// TwinCAT 3 PLC project InovanceDemo
// ProgramVersion: 3.1.4024.0
// libraries:
//   Tc2_MC2, * (Beckhoff Automation GmbH)
//   Tc2_Standard, * (Beckhoff Automation GmbH)
//   Tc2_System, * (Beckhoff Automation GmbH)
//   Tc3_Module, * (Beckhoff Automation GmbH)
// project tree:
//   DUTs/ MoveState.TcDUT
//   / PlcTask.TcTTO
//   POUs/ MAIN.TcPOU
// real-time tasks:
//   TASK PlcTask: cycle T#10ms, priority 20, ADS port 350
// motion (NC):
//   TASK NC-Task 1 SAF: cycle T#2ms, priority 4, ADS port 501
//   TASK NC-Task 1 SVB: cycle T#10ms, priority 8, ADS port 511
//   AXIS Axis 1 (id 1)
//     Velo: SlowManual=500
//     PositionAreaControl: Enable=false
//     TargetPosControl: Enable=false
//     OtherSettings: AllowMotionCmdToSlave=true
//     encoder EncType=1
//       EncPara: ScaleFactorNumerator=1.788e-05
//     drive DrvType=5
//       Analog: TorqueSetpointScale=10, ScaleFactorActTorque=0.1
//       TimeComp: TaskDelayCycles=1
//     controller CtrType=1
//       CtrPara: PriorControlFactor=1
//         PosDiffControl: Enable=false
//         Observer: BandWidth=20
// I/O:
//   DEVICE Device 3 (EtherCAT), AmsNetId 192.168.148.33.4.1
//     Drive 1 (InoSV660N) [SV660_1Axis_00915] (disabled)
// variable links:
//   InovanceDemo/InovanceDemo Instance <-> NC-Task 1 SAF/Axes/Axis 1
//     PlcTask Inputs/MAIN.Axis1.NcToPlc <-> Outputs/ToPlc
//     PlcTask Outputs/MAIN.Axis1.PlcToNc <-> Inputs/FromPlc

CONFIGURATION InovanceDemo
    RESOURCE PLC ON TwinCAT3
        TASK PlcTask(INTERVAL := T#10ms, PRIORITY := 20);
        PROGRAM MAIN WITH PlcTask : MAIN;
    END_RESOURCE
END_CONFIGURATION

// ---- DUTs/MoveState.TcDUT
TYPE MoveState :
(
	MOVE_INIT ,
	MOVE_ENABLE ,
	MOVE_MOVEFORWARD ,
	MOVE_MOVEBACKWARD ,
	MOVE_ERROR ,
	MOVE_RESET
)UDINT;
END_TYPE

// ---- POUs/MAIN.TcPOU
PROGRAM MAIN
VAR
	Axis1 : AXIS_REF;
	
	PowerAxis1 : MC_Power;
	PowerAxis1Out : ST_McOutputs;
	
	ResetAxis1 : MC_Reset;
	ResetAxis1Out : ST_McOutputs;
	
	MoveAxis1 : MC_MoveAbsolute();
	MoveAxis2 : MC_MoveAbsolute;
	MoveAbsolute1 : ST_McOutputs;
	MoveAbsolute2 : ST_McOutputs;
	
	
	state : MoveState;
	
END_VAR


	(* update the axis status at the beginning of each cycle *)
	Axis1();
	
	(* move axis using a state machine *)
	CASE state OF
		
		MOVE_INIT :
			MoveAxis1.Execute := FALSE;
			MoveAxis2.Execute := FALSE;
			ResetAxis1.Execute := FALSE;
			state := MOVE_ENABLE;
		
		MOVE_ENABLE:
			PowerAxis1.Enable := TRUE;
			PowerAxis1.Enable_Positive := TRUE;
			PowerAxis1.Enable_Negative := TRUE;
			IF PowerAxis1.Status THEN
				state := MOVE_MOVEFORWARD;
			ELSIF PowerAxis1.Error THEN	
				state := MOVE_ERROR;
			END_IF
		MOVE_MOVEFORWARD:
			MoveAxis1.Execute := TRUE;
			MoveAxis1.Position := 500;
			MoveAxis1.Velocity := 500;
			
			IF MoveAxis1.Error THEN
				state := MOVE_ERROR;
			ELSIF MoveAxis1.Done THEN
				MoveAxis1.Execute := FALSE;
				state := MOVE_MOVEBACKWARD;
			END_IF
			
		MOVE_MOVEBACKWARD:
			MoveAxis1.Execute := TRUE;
			MoveAxis1.Position := 0;
			MoveAxis1.Velocity := 500;
			
			IF MoveAxis1.Error THEN
				state := MOVE_ERROR;
			ELSIF MoveAxis1.Done THEN
				MoveAxis1.Execute := FALSE;
				state := MOVE_MOVEFORWARD;
			END_IF
		MOVE_ERROR:
			//DO nothing here
		MOVE_RESET:
			//DO nothing here
	END_CASE
	
	ActPower();	(* call the power function block *)
	ActMove();	(* call the move function block *)
	ActReset();	(* call the reset function block *)

ACTION ActMove:
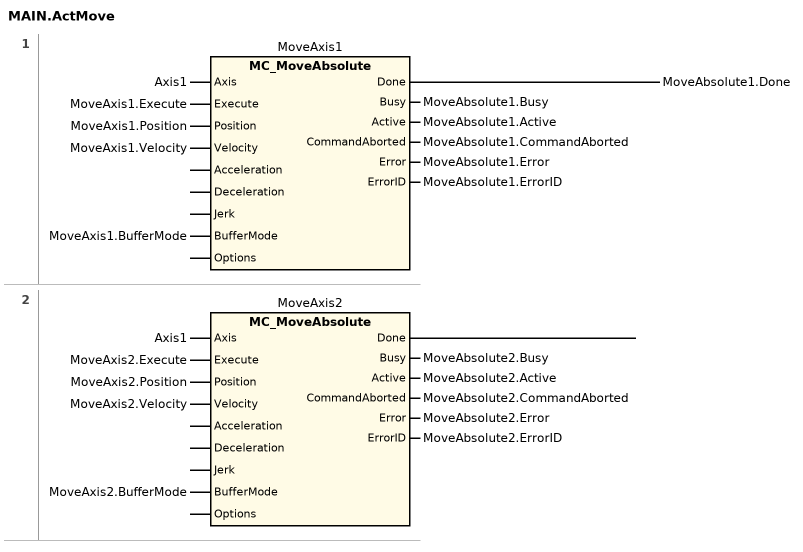
// NETWORK 1
MoveAxis1(
    Axis := Axis1,
    Execute := MoveAxis1.Execute,
    Position := MoveAxis1.Position,
    Velocity := MoveAxis1.Velocity,
    BufferMode := MoveAxis1.BufferMode,
    Busy => MoveAbsolute1.Busy,
    Active => MoveAbsolute1.Active,
    CommandAborted => MoveAbsolute1.CommandAborted,
    Error => MoveAbsolute1.Error,
    ErrorID => MoveAbsolute1.ErrorID); // MC_MoveAbsolute
MoveAbsolute1.Done := MoveAxis1.Done;

// NETWORK 2
MoveAxis2(
    Axis := Axis1,
    Execute := MoveAxis2.Execute,
    Position := MoveAxis2.Position,
    Velocity := MoveAxis2.Velocity,
    BufferMode := MoveAxis2.BufferMode,
    Busy => MoveAbsolute2.Busy,
    Active => MoveAbsolute2.Active,
    CommandAborted => MoveAbsolute2.CommandAborted,
    Error => MoveAbsolute2.Error,
    ErrorID => MoveAbsolute2.ErrorID); // MC_MoveAbsolute
END_ACTION

ACTION ActPower:
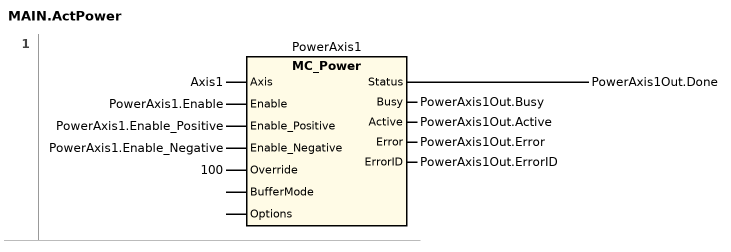
// NETWORK 1
PowerAxis1(
    Axis := Axis1,
    Enable := PowerAxis1.Enable,
    Enable_Positive := PowerAxis1.Enable_Positive,
    Enable_Negative := PowerAxis1.Enable_Negative,
    Override := 100,
    Busy => PowerAxis1Out.Busy,
    Active => PowerAxis1Out.Active,
    Error => PowerAxis1Out.Error,
    ErrorID => PowerAxis1Out.ErrorID); // MC_Power
PowerAxis1Out.Done := PowerAxis1.Status;
END_ACTION

ACTION ActReset:
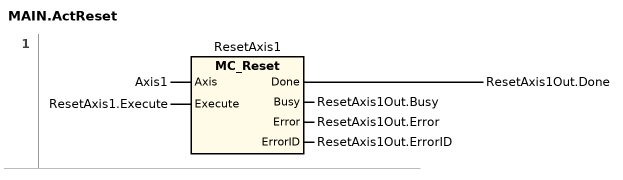
// NETWORK 1
ResetAxis1(
    Axis := Axis1,
    Execute := ResetAxis1.Execute,
    Busy => ResetAxis1Out.Busy,
    Error => ResetAxis1Out.Error,
    ErrorID => ResetAxis1Out.ErrorID); // MC_Reset
ResetAxis1Out.Done := ResetAxis1.Done;
END_ACTION

END_PROGRAM
